{attribute addProperty BoxType "EK1100-0000-0018"}
{attribute addProperty Id "Beckhoff_EL33xxEK1122Beckhoff_EL33xxEK1122_B04A0A54162A_0001_EL3311_0000_0016EL3311_4C36C06416821A_0002_EL3311_0000_0017EL3311_4C36C06416821A_0003_EL3311_0000_0018EL3311_18CEA68E12816A_0004_EL3311_0000_0019EL3311_18CEA68E12816A_0005_EL3311_0000_0020EL3311_18CEA68E12816A_0006_EL3311_0000_0021EL3311_18CEA68E12816A_0007_EL3311_0000_0022EL3311_18CEA68E12816A_0008_EL3311_0000_0023EL3311_18CEA68E12816A_0009_EL3312_0000_0016EL3312_FC0A385E24030A_0010_EL3312_0000_0017EL3312_FC0A385E24030A_0011_EL3312_0000_0018EL3312_322B585516020A_0012_EL3312_0000_0019EL3312_322B585516020A_0013_EL3312_0000_0020EL3312_322B585516020A_0014_EL3312_0000_0021EL3312_322B585516020A_0015_EL3312_0000_0022EL3312_322B585516020A_0016_EL3312_0000_0023EL3312_322B585516020A_0017_EL3314_0000_0016EL3314_483A859838448A_0018_EL3314_0000_0017EL3314_483A859838448A_0019_EL3314_0000_0018EL3314_00C6477622428A_0020_EL3314_0000_0019EL3314_00C6477622428A_0021_EL3314_0000_0020EL3314_00C6477622428A_0022_EL3314_0000_0021EL3314_00C6477622428A_0023_EL3314_0000_0022EL3314_00C6477622428A_0024_EL3314_0000_0023EL3314_00C6477622428A_0025_EL3314_0000_0024EL3314_00C6477622428A_0026_EL3314_0002_0016EL3314_43B876C128836A_0027_EL3314_0010_0016EL3314_2530FC3159674.5A_0028_EL3314_0010_0017EL3314_2530FC3159674.5A_0029_EL3314_0010_0018EL3314_1C7E98A428836A_0030_EL3314_0010_0019EL3314_1C7E98A428836A_0031_EL3314_0010_0020EL3314_645580BD28836A_0032_EL3314_0010_0021EL3314_645580BD28836A_0033_EL3314_0090_0016EL3314_2E54E3B022428A_0034_EL3314_0090_0017EL3314_2E54E3B022428A_0035_EL3318_0000_0016EL3318_B1CC74FF968121A_0036_EL3318_0000_0017EL3318_B1CC74FF968121A_0037_EL3318_0000_0018EL3318_B1CC74FF968121A_0038_EL3318_0000_0019EL3318_B1CC74FF968121A_0039_EL3318_0000_0020EL3318_B1CC74FF968121A_0040_EL3318_0000_0021EL3318_B1CC74FF968121A_0041_EL3318_0000_0022EL3318_B1CC74FF968121A_0042_EL3351_0000_0016EL3351_606039E324030A_0043_EL3351_0000_0017EL3351_606039E324030A_0044_EL3351_0000_0018EL3351_606039E324030A_0045_EL3351_0000_0019EL3351_606039E324030A_0046_EL3351_0000_0020EL3351_606039E324030A_0047_EL3356_0000_0017EL3356_D3F44C8116020A_0048_EL3356_0000_0018EL3356_D3F44C8116020A_0049_EL3356_0000_0019EL3356_D3F44C8116020A_0050_EL3356_0000_0020EL3356_D3F44C8116020A_0051_EL3356_0000_0021EL3356_E97824C816020A_0052_EL3356_0000_0022EL3356_E97824C816020A_0053_EL3356_0000_0023EL3356_E97824C816020A_0054_EL3356_0000_0024EL3356_E97824C816020A_0055_EL3356_0000_0025EL3356_E97824C816020A_0056_EL3356_0010_0017EL3356_F0DA284616020A_0057_EL3356_0010_0018EL3356_F0DA284616020A_0058_EL3356_0010_0019EL3356_F0DA284616020A_0059_EL3356_0010_0020EL3356_F0DA284616020A_0060_EL3356_0010_0021EL3356_CA56400F16020A_0061_EL3356_0010_0022EL3356_CA56400F16020A_0062_EL3356_0010_0023EL3356_CA56400F16020A_0063_EL3356_0010_0024EL3356_CA56400F16020A_0064_EL3356_0010_0025EL3356_CA56400F16020A_0065_EL3356_0020_0025EL3356_CA56400F16020A_0066_EL3356_0090_0025EL3356_CA56400F16020"}
{attribute addProperty CRC "1589309552"}
{attribute addProperty SizeInBites "19152"}
{attribute addProperty SizeInBytes "2394"}
TYPE Beckhoff_EL33xx_5EBAF070 EXTENDS EK1100_179A0949 :
STRUCT
	{attribute addProperty Name "Beckhoff_EL33xxEK1122"}
	Beckhoff_EL33xxEK1122 : Beckhoff_EL33xxEK1122_B04A0A54;
	{attribute addProperty Name "A_0001_EL3311_0000_0016"}
	A_0001_EL3311_0000_0016 : EL3311_4C36C064;
	{attribute addProperty Name "A_0002_EL3311_0000_0017"}
	A_0002_EL3311_0000_0017 : EL3311_4C36C064;
	{attribute addProperty Name "A_0003_EL3311_0000_0018"}
	A_0003_EL3311_0000_0018 : EL3311_18CEA68E;
	{attribute addProperty Name "A_0004_EL3311_0000_0019"}
	A_0004_EL3311_0000_0019 : EL3311_18CEA68E;
	{attribute addProperty Name "A_0005_EL3311_0000_0020"}
	A_0005_EL3311_0000_0020 : EL3311_18CEA68E;
	{attribute addProperty Name "A_0006_EL3311_0000_0021"}
	A_0006_EL3311_0000_0021 : EL3311_18CEA68E;
	{attribute addProperty Name "A_0007_EL3311_0000_0022"}
	A_0007_EL3311_0000_0022 : EL3311_18CEA68E;
	{attribute addProperty Name "A_0008_EL3311_0000_0023"}
	A_0008_EL3311_0000_0023 : EL3311_18CEA68E;
	{attribute addProperty Name "A_0009_EL3312_0000_0016"}
	A_0009_EL3312_0000_0016 : EL3312_FC0A385E;
	{attribute addProperty Name "A_0010_EL3312_0000_0017"}
	A_0010_EL3312_0000_0017 : EL3312_FC0A385E;
	{attribute addProperty Name "A_0011_EL3312_0000_0018"}
	A_0011_EL3312_0000_0018 : EL3312_322B5855;
	{attribute addProperty Name "A_0012_EL3312_0000_0019"}
	A_0012_EL3312_0000_0019 : EL3312_322B5855;
	{attribute addProperty Name "A_0013_EL3312_0000_0020"}
	A_0013_EL3312_0000_0020 : EL3312_322B5855;
	{attribute addProperty Name "A_0014_EL3312_0000_0021"}
	A_0014_EL3312_0000_0021 : EL3312_322B5855;
	{attribute addProperty Name "A_0015_EL3312_0000_0022"}
	A_0015_EL3312_0000_0022 : EL3312_322B5855;
	{attribute addProperty Name "A_0016_EL3312_0000_0023"}
	A_0016_EL3312_0000_0023 : EL3312_322B5855;
	{attribute addProperty Name "A_0017_EL3314_0000_0016"}
	A_0017_EL3314_0000_0016 : EL3314_483A8598;
	{attribute addProperty Name "A_0018_EL3314_0000_0017"}
	A_0018_EL3314_0000_0017 : EL3314_483A8598;
	{attribute addProperty Name "A_0019_EL3314_0000_0018"}
	A_0019_EL3314_0000_0018 : EL3314_00C64776;
	{attribute addProperty Name "A_0020_EL3314_0000_0019"}
	A_0020_EL3314_0000_0019 : EL3314_00C64776;
	{attribute addProperty Name "A_0021_EL3314_0000_0020"}
	A_0021_EL3314_0000_0020 : EL3314_00C64776;
	{attribute addProperty Name "A_0022_EL3314_0000_0021"}
	A_0022_EL3314_0000_0021 : EL3314_00C64776;
	{attribute addProperty Name "A_0023_EL3314_0000_0022"}
	A_0023_EL3314_0000_0022 : EL3314_00C64776;
	{attribute addProperty Name "A_0024_EL3314_0000_0023"}
	A_0024_EL3314_0000_0023 : EL3314_00C64776;
	{attribute addProperty Name "A_0025_EL3314_0000_0024"}
	A_0025_EL3314_0000_0024 : EL3314_00C64776;
	{attribute addProperty Name "A_0026_EL3314_0002_0016"}
	A_0026_EL3314_0002_0016 : EL3314_43B876C1;
	{attribute addProperty Name "A_0027_EL3314_0010_0016"}
	A_0027_EL3314_0010_0016 : EL3314_2530FC31;
	{attribute addProperty Name "A_0028_EL3314_0010_0017"}
	A_0028_EL3314_0010_0017 : EL3314_2530FC31;
	{attribute addProperty Name "A_0029_EL3314_0010_0018"}
	A_0029_EL3314_0010_0018 : EL3314_1C7E98A4;
	{attribute addProperty Name "A_0030_EL3314_0010_0019"}
	A_0030_EL3314_0010_0019 : EL3314_1C7E98A4;
	{attribute addProperty Name "A_0031_EL3314_0010_0020"}
	A_0031_EL3314_0010_0020 : EL3314_645580BD;
	{attribute addProperty Name "A_0032_EL3314_0010_0021"}
	A_0032_EL3314_0010_0021 : EL3314_645580BD;
	{attribute addProperty Name "A_0033_EL3314_0090_0016"}
	A_0033_EL3314_0090_0016 : EL3314_2E54E3B0;
	{attribute addProperty Name "A_0034_EL3314_0090_0017"}
	A_0034_EL3314_0090_0017 : EL3314_2E54E3B0;
	{attribute addProperty Name "A_0035_EL3318_0000_0016"}
	A_0035_EL3318_0000_0016 : EL3318_B1CC74FF;
	{attribute addProperty Name "A_0036_EL3318_0000_0017"}
	A_0036_EL3318_0000_0017 : EL3318_B1CC74FF;
	{attribute addProperty Name "A_0037_EL3318_0000_0018"}
	A_0037_EL3318_0000_0018 : EL3318_B1CC74FF;
	{attribute addProperty Name "A_0038_EL3318_0000_0019"}
	A_0038_EL3318_0000_0019 : EL3318_B1CC74FF;
	{attribute addProperty Name "A_0039_EL3318_0000_0020"}
	A_0039_EL3318_0000_0020 : EL3318_B1CC74FF;
	{attribute addProperty Name "A_0040_EL3318_0000_0021"}
	A_0040_EL3318_0000_0021 : EL3318_B1CC74FF;
	{attribute addProperty Name "A_0041_EL3318_0000_0022"}
	A_0041_EL3318_0000_0022 : EL3318_B1CC74FF;
	{attribute addProperty Name "A_0042_EL3351_0000_0016"}
	A_0042_EL3351_0000_0016 : EL3351_606039E3;
	{attribute addProperty Name "A_0043_EL3351_0000_0017"}
	A_0043_EL3351_0000_0017 : EL3351_606039E3;
	{attribute addProperty Name "A_0044_EL3351_0000_0018"}
	A_0044_EL3351_0000_0018 : EL3351_606039E3;
	{attribute addProperty Name "A_0045_EL3351_0000_0019"}
	A_0045_EL3351_0000_0019 : EL3351_606039E3;
	{attribute addProperty Name "A_0046_EL3351_0000_0020"}
	A_0046_EL3351_0000_0020 : EL3351_606039E3;
	{attribute addProperty Name "A_0047_EL3356_0000_0017"}
	A_0047_EL3356_0000_0017 : EL3356_D3F44C81;
	{attribute addProperty Name "A_0048_EL3356_0000_0018"}
	A_0048_EL3356_0000_0018 : EL3356_D3F44C81;
	{attribute addProperty Name "A_0049_EL3356_0000_0019"}
	A_0049_EL3356_0000_0019 : EL3356_D3F44C81;
	{attribute addProperty Name "A_0050_EL3356_0000_0020"}
	A_0050_EL3356_0000_0020 : EL3356_D3F44C81;
	{attribute addProperty Name "A_0051_EL3356_0000_0021"}
	A_0051_EL3356_0000_0021 : EL3356_E97824C8;
	{attribute addProperty Name "A_0052_EL3356_0000_0022"}
	A_0052_EL3356_0000_0022 : EL3356_E97824C8;
	{attribute addProperty Name "A_0053_EL3356_0000_0023"}
	A_0053_EL3356_0000_0023 : EL3356_E97824C8;
	{attribute addProperty Name "A_0054_EL3356_0000_0024"}
	A_0054_EL3356_0000_0024 : EL3356_E97824C8;
	{attribute addProperty Name "A_0055_EL3356_0000_0025"}
	A_0055_EL3356_0000_0025 : EL3356_E97824C8;
	{attribute addProperty Name "A_0056_EL3356_0010_0017"}
	A_0056_EL3356_0010_0017 : EL3356_F0DA2846;
	{attribute addProperty Name "A_0057_EL3356_0010_0018"}
	A_0057_EL3356_0010_0018 : EL3356_F0DA2846;
	{attribute addProperty Name "A_0058_EL3356_0010_0019"}
	A_0058_EL3356_0010_0019 : EL3356_F0DA2846;
	{attribute addProperty Name "A_0059_EL3356_0010_0020"}
	A_0059_EL3356_0010_0020 : EL3356_F0DA2846;
	{attribute addProperty Name "A_0060_EL3356_0010_0021"}
	A_0060_EL3356_0010_0021 : EL3356_CA56400F;
	{attribute addProperty Name "A_0061_EL3356_0010_0022"}
	A_0061_EL3356_0010_0022 : EL3356_CA56400F;
	{attribute addProperty Name "A_0062_EL3356_0010_0023"}
	A_0062_EL3356_0010_0023 : EL3356_CA56400F;
	{attribute addProperty Name "A_0063_EL3356_0010_0024"}
	A_0063_EL3356_0010_0024 : EL3356_CA56400F;
	{attribute addProperty Name "A_0064_EL3356_0010_0025"}
	A_0064_EL3356_0010_0025 : EL3356_CA56400F;
	{attribute addProperty Name "A_0065_EL3356_0020_0025"}
	A_0065_EL3356_0020_0025 : EL3356_CA56400F;
	{attribute addProperty Name "A_0066_EL3356_0090_0025"}
	A_0066_EL3356_0090_0025 : EL3356_CA56400F;
END_STRUCT
END_TYPE

(* stored: Version 1.2.0.0, ProductVersion 3.1.4024.9
   DUT Beckhoff_EL33xx_5EBAF070: Id {f37c1324-7065-4ad4-9821-461800dd9f40} *)
